(* CoDeSys 2.3.9.37 project: Cap12_6.pro *)
(* Libraries: Standard.lib 4.10.05 12:14:46 *)

(* POU PLC_PRG, FBD *)
PROGRAM PLC_PRG
VAR
	MiPWM: PWM;
       Valor: REAL;
	Sal: BOOL;
END_VAR
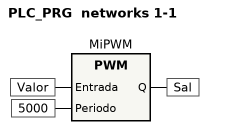
_FBD_ (* Function Block Diagram *)
NETWORK 1
	MiPWM:PWM(Entrada: Valor, Periodo: 5000) => Sal
_END_FBD_
(* the same logic as Structured Text *)
(* Network 1 *)
MiPWM(Entrada := Valor, Periodo := 5000);
Sal := MiPWM.Q;
END_PROGRAM

(* POU PWM, ST *)
FUNCTION_BLOCK PWM
VAR_INPUT
      Entrada :REAL;
      Periodo: REAL := 100;
END_VAR
VAR_OUTPUT
     Q : BOOL;
END_VAR
VAR
	tact: TIME;      (* Instante de tiempo actual *)
	MiPulso: Pulso;   (* Instancia de tipo Pulso *)
	Flanco: BOOL;   (* Detección de comienzo periodo*)
	Comienzo: TIME; (* Almacena el instante en que comenzó el periodo *)
	Intervalo: TIME; (* Tiempo transcurrido desde que comenzó el periodo actual *)
	TiempoUP: TIME;  (*Tiempo en que la señal está a 1 *)
END_VAR
tact:=TIME();
(* Detecta el comienzo del periodo *)
MiPulso(Periodo:=Periodo, Salida=>Flanco);
(* Calcula el intervalo en que la salida está a 1 *)
TiempoUP:=REAL_TO_TIME(Entrada*Periodo);

IF Flanco THEN
   Comienzo:=tact;
   Q:= TiempoUP > T#0ms;
ELSIF Q THEN
    Intervalo:=tact-Comienzo;
    IF Intervalo >= TiempoUP THEN
          Q:=FALSE;
          Intervalo:=T#0ms;
    END_IF
END_IF
END_FUNCTION_BLOCK

(* POU Pulso, ST *)
FUNCTION_BLOCK Pulso
VAR_INPUT
     Periodo : REAL:=100;
END_VAR
VAR_OUTPUT
    Salida : BOOL;
END_VAR
VAR
	tact: TIME;    (*Instante de tiempo actual *)
	Ciclo1: BOOL:=TRUE;  (* Ejecución delprimer ciclo del PLC *)
	told: TIME;     (* Instante de tiempo en que se produjo el último pulso *)
	TiempoPulso: TIME;    (* Periodo en formato TIME *)
END_VAR
tact:=TIME();
TiempoPulso:=REAL_TO_TIME(Periodo);

IF Ciclo1 THEN
  Ciclo1 := FALSE;
   told := tact-TiempoPulso;
END_IF

Salida:=tact-told >=TiempoPulso;
IF Salida THEN
  told := tact;
END_IF
END_FUNCTION_BLOCK

(* Visualisation Visu
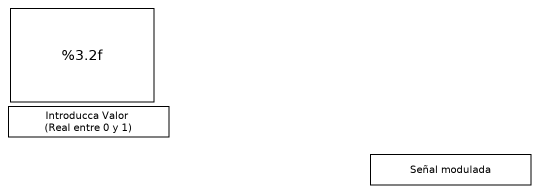
rectangle at (44,98)-(188,192): text "%3.2f"; shows PLC_PRG.Valor; editable 0..1
rectangle at (42,196)-(203,227): text "Introducca Valor / (Real entre 0 y 1)"
rectangle at (404,244)-(565,275): text "Señal modulada"
1 elements of other kinds (tables, trends, ...) not read
*)
